FUNCTION_BLOCK Merging (* Template for a Basic Function Block Type *)
  (* Standard: 61499-2 *)
  (* Version 1.0, 2023-10-14, ADMIN *)
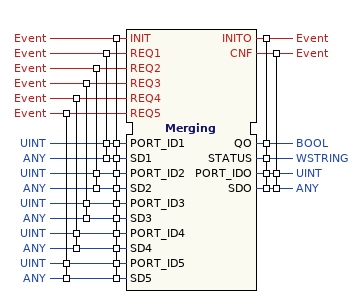
  EVENT_INPUT
    INIT WITH PORT_ID1, SD1, PORT_ID2, SD2, PORT_ID3, SD3, PORT_ID4, SD4, PORT_ID5, SD5; (* Initialization Request *)
    REQ1 WITH PORT_ID1, SD1; (* Normal Execution Request *)
    REQ2 WITH PORT_ID2, SD2;
    REQ3 WITH PORT_ID3, SD3;
    REQ4 WITH PORT_ID4, SD4;
    REQ5 WITH PORT_ID5, SD5;
  END_EVENT
  EVENT_OUTPUT
    INITO WITH QO, STATUS, PORT_IDO, SDO; (* Initialization Confirm *)
    CNF WITH PORT_IDO, SDO; (* Execution Confirmation *)
  END_EVENT
  VAR_INPUT
    PORT_ID1 : UINT; (* Port ID 1 *)
    SD1 : ANY;
    PORT_ID2 : UINT; (* Port ID 2 *)
    SD2 : ANY;
    PORT_ID3 : UINT; (* Port ID 3 *)
    SD3 : ANY;
    PORT_ID4 : UINT; (* Port ID 4 *)
    SD4 : ANY;
    PORT_ID5 : UINT; (* Port ID 5 *)
    SD5 : ANY;
  END_VAR
  VAR_OUTPUT
    QO : BOOL; (* Output event qualifier *)
    STATUS : WSTRING; (* Service Status *)
    PORT_IDO : UINT; (* Port ID Out *)
    SDO : ANY;
  END_VAR
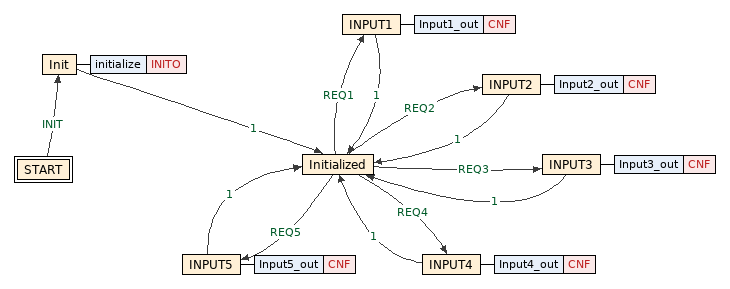
  EC_STATES
    START; (* Initial State *)
    Init : initialize -> INITO; (* Initialization *)
    INPUT1 : Input1_out -> CNF; (* Normal execution *)
    Initialized;
    INPUT2 : Input2_out -> CNF;
    INPUT3 : Input3_out -> CNF;
    INPUT4 : Input4_out -> CNF;
    INPUT5 : Input5_out -> CNF;
  END_STATES
  EC_TRANSITIONS
    START TO Init := INIT;
    Init TO Initialized := 1;
    Initialized TO INPUT1 := REQ1;
    INPUT1 TO Initialized := 1;
    Initialized TO INPUT2 := REQ2;
    INPUT2 TO Initialized := 1;
    Initialized TO INPUT3 := REQ3;
    INPUT3 TO Initialized := 1;
    Initialized TO INPUT4 := REQ4;
    INPUT4 TO Initialized := 1;
    Initialized TO INPUT5 := REQ5;
    INPUT5 TO Initialized := 1;
  END_TRANSITIONS
  ALGORITHM initialize IN ST: (* Initialization algorithm *)

  END_ALGORITHM
  ALGORITHM deInitialize IN ST: (* Normally executed algorithm *)
QO := FALSE;
  END_ALGORITHM
  ALGORITHM Input1_out IN ST:
QO := 1;
STATUS := "NORMAL";

PORT_IDO := PORT_ID1;
SDO := SD1;
  END_ALGORITHM
  ALGORITHM Input3_out IN ST:
QO := 1;
STATUS := "NORMAL";

PORT_IDO := PORT_ID3;
SDO := SD3;
  END_ALGORITHM
  ALGORITHM Input2_out IN ST:
QO := 1;
STATUS := "NORMAL";

PORT_IDO := PORT_ID2;
SDO := SD2;
  END_ALGORITHM
  ALGORITHM Input4_out IN ST:
QO := 1;
STATUS := "NORMAL";

PORT_IDO := PORT_ID4;
SDO := SD4;
  END_ALGORITHM
  ALGORITHM Input5_out IN ST:
QO := 1;
STATUS := "NORMAL";

PORT_IDO := PORT_ID5;
SDO := SD5;
  END_ALGORITHM
END_FUNCTION_BLOCK
